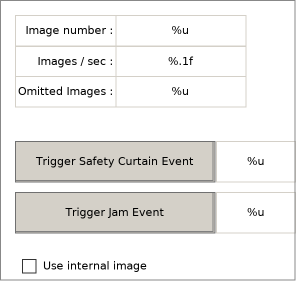
VISUALIZATION Visualization  // 296x281
    Textfield (115,15 131x31), "%u", text variable: Vision1.nImage_ID_Num
    Textfield (15,15 101x31), "Image number :", tooltip "Image number assigned by the camera."
    Textfield (115,46 131x31), "%.1f", text variable: Vision1.ImagePerSec
    Textfield (15,46 101x31), "Images / sec :"
    Button (15,141 200x41), "Trigger Safety Curtain Event"
        tap Vision1.TriggerEvent1
    Textfield (216,141 80x41), "%u", text variable: Vision1.CountEventTrigger1
    Textfield (115,76 131x31), "%u", text variable: Vision1.nImagesOmitted
    Textfield (15,76 101x31), "Omitted Images :", tooltip "Image number assigned by the camera."
    Checkbox (20,251 150x30), "Use internal image", variable: Vision1.UseCreatedTestImage
    Button (15,192 200x41), "Trigger Jam Event"
        tap Vision1.TriggerEvent2
    Textfield (216,192 80x41), "%u", text variable: Vision1.CountEventTrigger2
END_VISUALIZATION

(* stored: Version 1.1.0.1, ProductVersion 3.1.4026.13
   Visu Visualization: Id {32859f03-c167-45d3-b13a-7e57fa8c6398} *)
